INTERFACE I_CyclicTask EXTENDS __SYSTEM.IQueryInterface

METHOD Run
VAR_INPUT
END_VAR
END_METHOD

END_INTERFACE

(* stored: Version 1.1.0.1, ProductVersion 3.1.4024.12
   Itf I_CyclicTask: Id {474f2a5a-80bd-41d9-948d-26247a1ce276}
   Method Run: Id {676981b5-670e-448f-a624-da6140f640f1} *)
